FUNCTION_BLOCK carride
VAR_INPUT
    bStart : BOOL;
    TravelTime : TIME;
END_VAR

VAR_OUTPUT
    bcarArrived : BOOL := FALSE;
END_VAR

VAR
	tTimerauto :ton := (PT := T#8S); // timer auto
END_VAR

IF bStart AND NOT gvl.InternalStart THEN
    gvl.InternalStart := TRUE;
    bcarArrived := FALSE;
    tTimerauto(IN := TRUE, PT := TravelTime);
END_IF;

tTimerauto(IN := tTimerauto.IN, PT := TravelTime);


IF tTimerauto.Q THEN
    bcarArrived := TRUE;
    tTimerauto(IN := FALSE);
    gvl.InternalStart := FALSE;
END_IF;

END_FUNCTION_BLOCK

(* stored: Version 1.1.0.1, ProductVersion 3.1.4024.15
   POU carride: Id {1113fe9e-cd66-49f9-a801-011964240413}, SpecialFunc None *)
